FUNCTION_BLOCK EL3011
VAR
	_io : EL3xx1_Data;
	{attribute addProperty Name "WcState"}
	_wcState : WcStateInputToggle;
	{attribute addProperty Name "Info data"}
	_infoData : InfoDataAds;
END_VAR

PROPERTY IO : REFERENCE TO EL3xx1_Data
GET
IO REF= _io;
END_GET
END_PROPERTY

PROPERTY WcState : REFERENCE TO WcStateInputToggle
GET
WcState REF= _wcState;
END_GET
END_PROPERTY

END_FUNCTION_BLOCK

(* stored: Version 1.1.0.1, ProductVersion 3.1.4024.9
   POU EL3011: Id {84ebe98e-0882-0cf7-0312-c6dad1fa0843}, SpecialFunc None
   Property IO: Id {9149f5ae-060a-0eb1-0e17-7d3bc4ad680d}
   Get Get: Id {4121af79-368c-0bd4-0e3f-91c9d23ca5b5}
   Property WcState: Id {ae50bdbf-aea6-044e-11fe-fbe2bb47b276}
   Get Get: Id {df5b5955-4130-0572-1868-ff3b81f96ed4} *)
